% RSLogix 500 project LVD191219v4_Bot.RSS, saved by version 12.00.00.00 %
PROJECT "XLTCEBOT"    % processor: MicroLogix 1400 %

PROGRAM FILES
  LAD 2 "MAIN"  48 rungs  % Main Program Routine %
  LAD 4 "PACKAGER"  27 rungs  % normal %
  LAD 5 "NO PACKAGE"  7 rungs
  LAD 6 "TIMING"  11 rungs
  LAD 12 "ENABLES"  14 rungs
  LAD 14 "SPEED OUT"  14 rungs
  LAD 16 "TOTALCOUNT"  4 rungs
  LAD 18 "TESTTRIG1"  4 rungs
  LAD 20 "TESTTRIG2"  4 rungs
  LAD 24 "SKIPPED"  5 rungs
  LAD 70 "ALIGNFAILS"  4 rungs  % normal %
  LAD 80 "HSC BOT"  5 rungs
  LAD 100 "1 MS STI"  17 rungs  % high speed %
  LAD 102 "SPEED BOT"  8 rungs  % high speed %
  LAD 104 "P BOT"  7 rungs  % high speed %
  LAD 110 "SHIFT BOT"  7 rungs
  LAD 120 "OLDBOTOP"  7 rungs
  LAD 121 "OLDBOTOP"  8 rungs
  LAD 123 "BOTOPTIC"  2 rungs
  LAD 124 "BOTOPTIC"  4 rungs
  LAD 130 "INS1"  20 rungs
  LAD 131 "INS1RESULT"  7 rungs
  LAD 132 "INS1PASS"  5 rungs
  LAD 133 "INS1FAIL"  3 rungs
  LAD 134 "INS1ACQ"  8 rungs
  LAD 135 "Q1TIMETEST"  7 rungs
  LAD 136 "INS1TRIG"  6 rungs
  LAD 137 "FIFO1SET"  9 rungs
  LAD 138 "FIFO1GET"  8 rungs
  LAD 139 "INSDATA1"  3 rungs  % used for analysis %
  LAD 140 "TESTFAULT1"  9 rungs
  LAD 141 "INS1FIX1"  6 rungs
  LAD 142 "INS1FIX2"  3 rungs
  LAD 145 "INS2"  22 rungs
  LAD 146 "INS2RESULT"  7 rungs
  LAD 147 "INS2PASS"  5 rungs
  LAD 148 "INS2FAIL"  3 rungs
  LAD 149 "INS2ACQ"  8 rungs
  LAD 150 "Q2TIMETEST"  6 rungs
  LAD 151 "INS2TRIG"  5 rungs
  LAD 152 "FIFO2SET"  9 rungs
  LAD 153 "FIFO2GET"  8 rungs
  LAD 154 "INSDATA2"  3 rungs  % used for analysis %
  LAD 155 "TESTFAULT2"  9 rungs
  LAD 156 "INS2FIX1"  6 rungs
  LAD 157 "INS2FIX2"  3 rungs
  LAD 200 "XFEROUT"  9 rungs
  LAD 201 "XFER GOOD"  5 rungs
  LAD 202 "XFER NG"  5 rungs
  LAD 111, 122, 125, 144, 159: only END

DATA FILES
  O0 OUTPUT  11 elements
  I1 INPUT  11 elements
  S2 STATUS  66 elements
  B3 BINARY  64 elements
  T4 TIMER  40 elements
  C5 COUNTER  1 elements
  R6 CONTROL  20 elements
  N7 INTEGER  200 elements
  F8 FLOAT  100 elements
  B9 NU  256 elements
  B10 NU  1 elements
  B11 NU  256 elements
  B12 HMI_BINARY  22 elements  % general use with hmi to avoid additional reads %
  L13  COUNTS  256 elements
  F14 HMI_FLOATS  100 elements
  N15 HMI_INTS  100 elements
  L16 NU  100 elements
  B17 NU  128 elements
  B18 NU  128 elements
  L19 NU  10 elements
  L20 NU  10 elements
  L21 NU  10 elements
  L22 NU  10 elements
  L23 NU  100 elements
  L24 NU  100 elements
  L25 NU  10 elements
  L26 NU  10 elements
  L27 RATETIMES  50 elements  % Must have it's own file because it uses all 50 int %
  L28 INS1TIME  50 elements
  L29 INS1POS  50 elements
  L30 INS2TIME  50 elements
  L31 INS2POS  50 elements
  L42 COMS  52 elements
  RI43 RI1  11 elements
  MG44 MSG  11 elements
  B181 BLANK  256 elements  % used to wipe bs files %
  F182 TEST FLOAT  50 elements
  L183 TEST LONG  50 elements
  N184 TEST INTS  50 elements
  B185 TEST BITS  50 elements
  N186 HMI INTS  50 elements
  L187 HMI LONG  50 elements
  F188 HMI FLOAT  50 elements
  B189 HMI BITS  50 elements
  L190 COUNTS  50 elements
  B191 ERROR BITS  10 elements
  L192 SPD OFFSET  50 elements
  F193 SPD OFFSET  50 elements
  B194 BOT GOOD  128 elements
  B195 BOT NG  128 elements
  B196 CTRL BITS  50 elements
  N197 CTRL INTS  50 elements
  B198 TRK BITS  50 elements
  L199 TRK LONG  50 elements
  N200 TRK INTS  50 elements
  L201 INS LONG  50 elements
  B202 INS BITS  50 elements
  N203 INS INTS  50 elements
  L204 CTRL LONG  50 elements
  F205 CTRL FLTS  50 elements

LADDER 2 "MAIN"    % Main Program Routine %
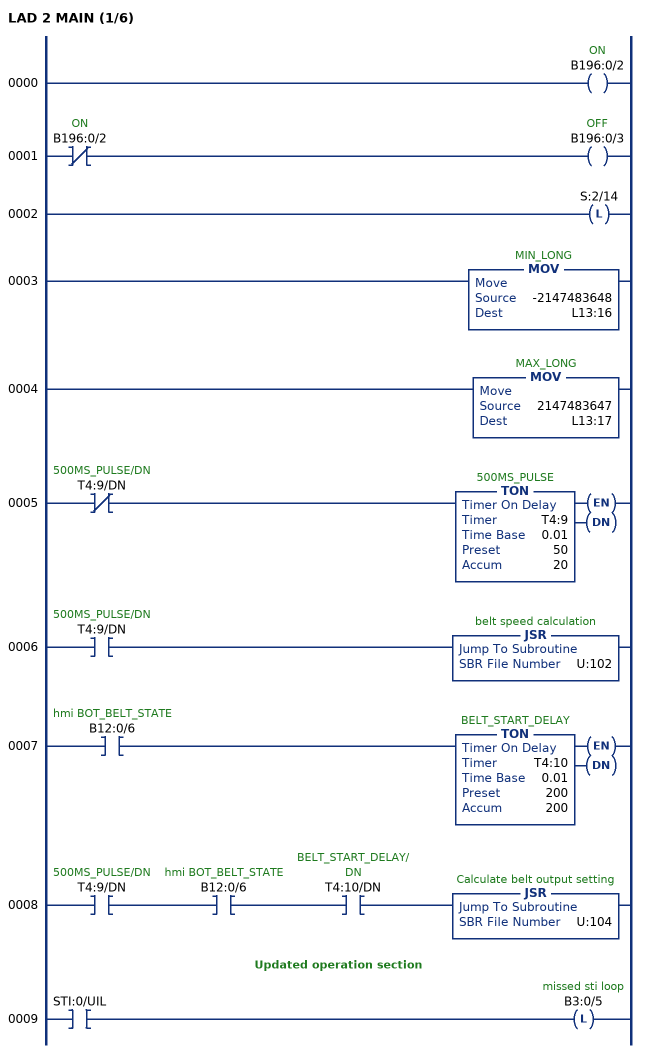
% Rung: 0 %
SOR OTE B196:0/2 EOR
%   B196:0/2  ON %
% Rung: 1 %
SOR XIO B196:0/2 OTE B196:0/3 EOR
%   B196:0/2  ON %
%   B196:0/3  OFF %
% Rung: 2 %
SOR OTL S:2/14 EOR
% Rung: 3 %
SOR MOV -2147483648 L13:16 EOR
%   L13:16  MIN_LONG %
% Rung: 4 %
SOR MOV 2147483647 L13:17 EOR
%   L13:17  MAX_LONG %
% Rung: 5 %
SOR XIO T4:9/DN TON T4:9 0.01 50 20 EOR
%   T4:9  500MS_PULSE %
% Rung: 6 %
SOR XIC T4:9/DN JSR U:102 EOR
%   T4:9  500MS_PULSE %
%   U:102  "belt speed calculation" %
% Rung: 7 %
SOR XIC B12:0/6 TON T4:10 0.01 200 200 EOR
%   B12:0/6  BOT_BELT_STATE  "hmi" %
%   T4:10  BELT_START_DELAY %
% Rung: 8 %
SOR XIC T4:9/DN XIC B12:0/6 XIC T4:10/DN JSR U:104 EOR
%   T4:9  500MS_PULSE %
%   B12:0/6  BOT_BELT_STATE  "hmi" %
%   T4:10  BELT_START_DELAY %
%   U:104  "Calculate belt output setting" %
% Rung: 9 %
% TITLE: Updated operation section %
SOR XIC STI:0/UIL OTL B3:0/5 EOR
%   B3:0/5  "missed sti loop" %

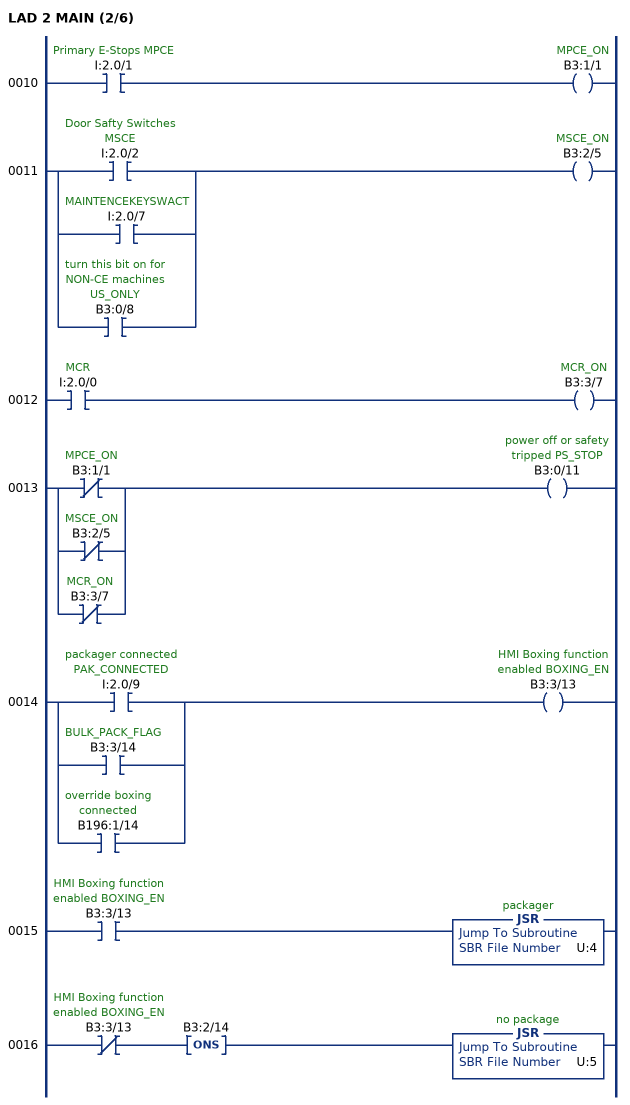
% Rung: 10 %
SOR XIC I:2.0/1 OTE B3:1/1 EOR
%   I:2.0/1  MPCE  "Primary E-Stops" %
%   B3:1/1  MPCE_ON %
% Rung: 11 %
SOR BST XIC I:2.0/2 NXB XIC I:2.0/7 NXB XIC B3:0/8 BND OTE B3:2/5 EOR
%   I:2.0/2  MSCE  "Door Safty Switches" %
%   I:2.0/7  MAINTENCEKEYSWACT %
%   B3:0/8  US_ONLY  "turn this bit on for NON-CE machines" %
%   B3:2/5  MSCE_ON %
% Rung: 12 %
SOR XIC I:2.0/0 OTE B3:3/7 EOR
%   I:2.0/0  MCR %
%   B3:3/7  MCR_ON %
% Rung: 13 %
SOR BST XIO B3:1/1 NXB XIO B3:2/5 NXB XIO B3:3/7 BND OTE B3:0/11 EOR
%   B3:1/1  MPCE_ON %
%   B3:2/5  MSCE_ON %
%   B3:3/7  MCR_ON %
%   B3:0/11  PS_STOP  "power off or safety tripped" %
% Rung: 14 %
SOR BST XIC I:2.0/9 NXB XIC B3:3/14 NXB XIC B196:1/14 BND OTE B3:3/13 EOR
%   I:2.0/9  PAK_CONNECTED  "packager connected" %
%   B3:3/14  BULK_PACK_FLAG %
%   B196:1/14  "override boxing connected" %
%   B3:3/13  BOXING_EN  "HMI Boxing function enabled" %
% Rung: 15 %
SOR XIC B3:3/13 JSR U:4 EOR
%   B3:3/13  BOXING_EN  "HMI Boxing function enabled" %
%   U:4  "packager" %
% Rung: 16 %
SOR XIO B3:3/13 ONS B3:2/14 JSR U:5 EOR
%   B3:3/13  BOXING_EN  "HMI Boxing function enabled" %
%   U:5  "no package" %

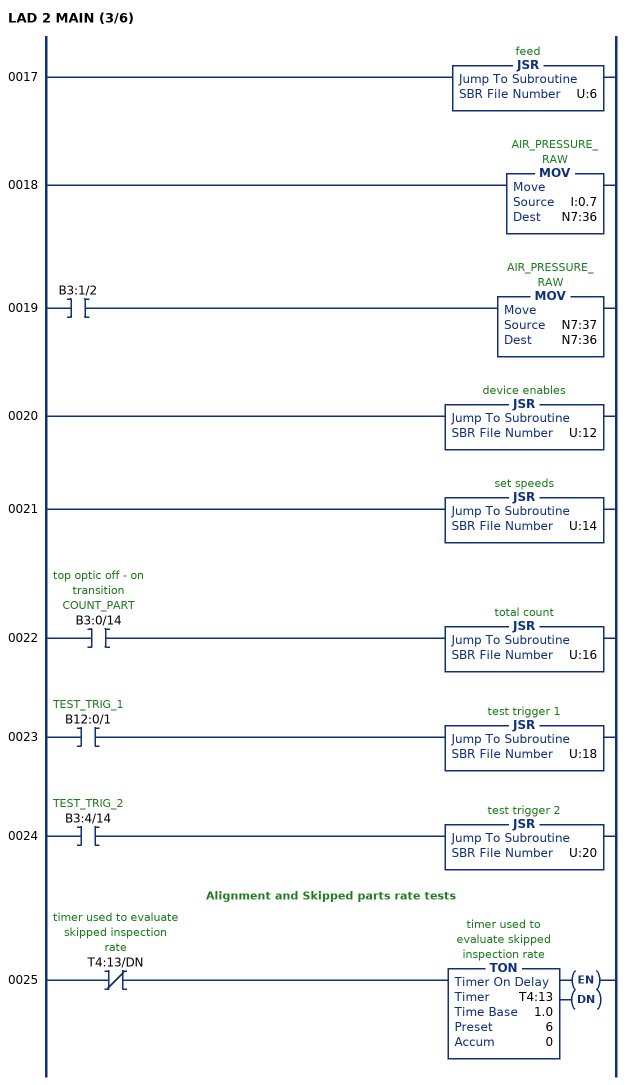
% Rung: 17 %
SOR JSR U:6 EOR
%   U:6  "feed" %
% Rung: 18 %
SOR MOV I:0.7 N7:36 EOR
%   I:0.7  AIR_PRESSURE  "Air Presure Sensor Input Signal" %
%   N7:36  AIR_PRESSURE_RAW %
% Rung: 19 %
SOR XIC B3:1/2 MOV N7:37 N7:36 EOR
%   N7:36  AIR_PRESSURE_RAW %
% Rung: 20 %
SOR JSR U:12 EOR
%   U:12  "device enables" %
% Rung: 21 %
SOR JSR U:14 EOR
%   U:14  "set speeds" %
% Rung: 22 %
SOR XIC B3:0/14 JSR U:16 EOR
%   B3:0/14  COUNT_PART  "top optic off - on transition" %
%   U:16  "total count" %
% Rung: 23 %
SOR XIC B12:0/1 JSR U:18 EOR
%   B12:0/1  TEST_TRIG_1 %
%   U:18  "test trigger 1" %
% Rung: 24 %
SOR XIC B3:4/14 JSR U:20 EOR
%   B3:4/14  TEST_TRIG_2 %
%   U:20  "test trigger 2" %
% Rung: 25 %
% TITLE: Alignment and Skipped parts rate tests %
SOR XIO T4:13/DN TON T4:13 1.0 6 0 EOR
%   T4:13  "timer used to evaluate skipped inspection rate" %

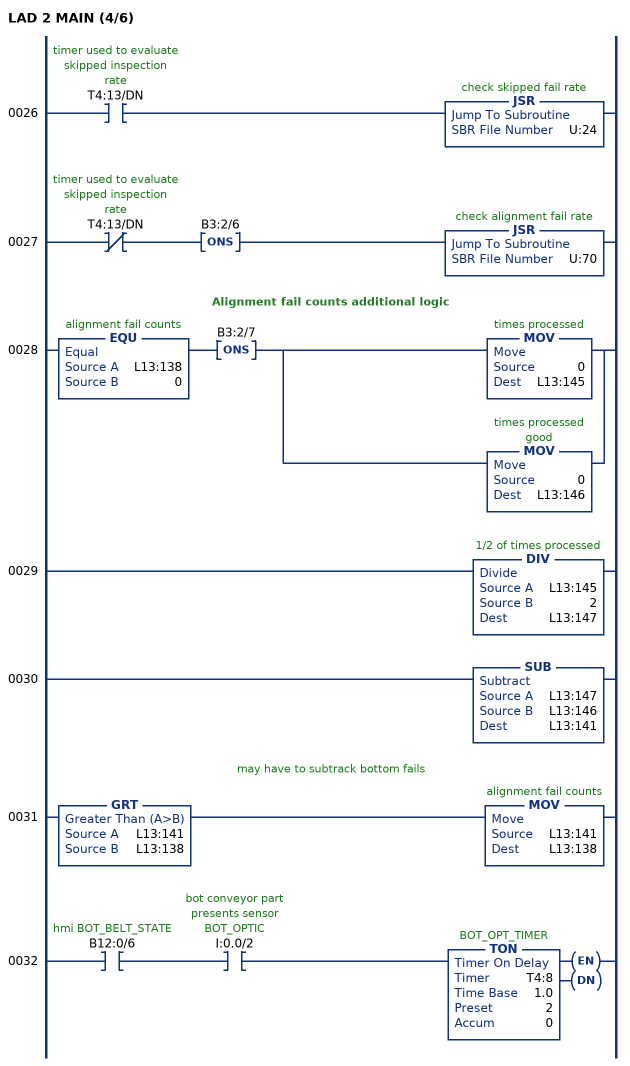
% Rung: 26 %
SOR XIC T4:13/DN JSR U:24 EOR
%   T4:13  "timer used to evaluate skipped inspection rate" %
%   U:24  "check skipped fail rate" %
% Rung: 27 %
SOR XIO T4:13/DN ONS B3:2/6 JSR U:70 EOR
%   T4:13  "timer used to evaluate skipped inspection rate" %
%   U:70  "check alignment fail rate" %
% Rung: 28 %
% TITLE: Alignment fail counts additional logic %
SOR EQU L13:138 0 ONS B3:2/7 BST MOV 0 L13:145 NXB MOV 0 L13:146 BND EOR
%   L13:138  "alignment fail counts" %
%   L13:145  "times processed" %
%   L13:146  "times processed good" %
% Rung: 29 %
SOR DIV L13:145 2 L13:147 EOR
%   L13:145  "times processed" %
%   L13:147  "1/2 of times processed" %
% Rung: 30 %
SOR SUB L13:147 L13:146 L13:141 EOR
%   L13:147  "1/2 of times processed" %
%   L13:146  "times processed good" %
% Rung: 31 %
% may have to subtrack bottom fails %
SOR GRT L13:141 L13:138 MOV L13:141 L13:138 EOR
%   L13:138  "alignment fail counts" %
% Rung: 32 %
SOR XIC B12:0/6 XIC I:0.0/2 TON T4:8 1.0 2 0 EOR
%   B12:0/6  BOT_BELT_STATE  "hmi" %
%   I:0.0/2  BOT_OPTIC  "bot conveyor part presents sensor" %
%   T4:8  BOT_OPT_TIMER %

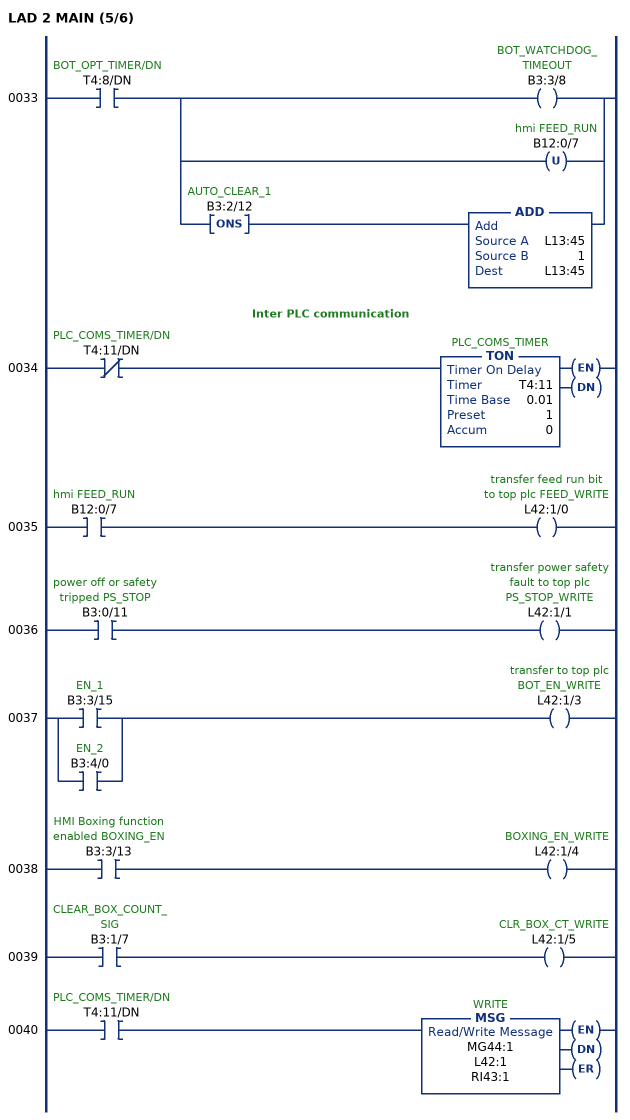
% Rung: 33 %
SOR XIC T4:8/DN BST OTE B3:3/8 NXB OTU B12:0/7 NXB ONS B3:2/12 ADD L13:45 1 L13:45 BND EOR
%   T4:8  BOT_OPT_TIMER %
%   B3:3/8  BOT_WATCHDOG_TIMEOUT %
%   B12:0/7  FEED_RUN  "hmi" %
%   B3:2/12  AUTO_CLEAR_1 %
% Rung: 34 %
% TITLE: Inter PLC communication %
SOR XIO T4:11/DN TON T4:11 0.01 1 0 EOR
%   T4:11  PLC_COMS_TIMER %
% Rung: 35 %
SOR XIC B12:0/7 OTE L42:1/0 EOR
%   B12:0/7  FEED_RUN  "hmi" %
%   L42:1/0  FEED_WRITE  "transfer feed run bit to top plc" %
% Rung: 36 %
SOR XIC B3:0/11 OTE L42:1/1 EOR
%   B3:0/11  PS_STOP  "power off or safety tripped" %
%   L42:1/1  PS_STOP_WRITE  "transfer power safety fault to top plc" %
% Rung: 37 %
SOR BST XIC B3:3/15 NXB XIC B3:4/0 BND OTE L42:1/3 EOR
%   B3:3/15  EN_1 %
%   B3:4/0  EN_2 %
%   L42:1/3  BOT_EN_WRITE  "transfer to top plc" %
% Rung: 38 %
SOR XIC B3:3/13 OTE L42:1/4 EOR
%   B3:3/13  BOXING_EN  "HMI Boxing function enabled" %
%   L42:1/4  BOXING_EN_WRITE %
% Rung: 39 %
SOR XIC B3:1/7 OTE L42:1/5 EOR
%   B3:1/7  CLEAR_BOX_COUNT_SIG %
%   L42:1/5  CLR_BOX_CT_WRITE %
% Rung: 40 %
SOR XIC T4:11/DN MSG MG44:1 L42:1 RI43:1 EOR
%   T4:11  PLC_COMS_TIMER %
%   MSG set-up: 500CPU Write | 33 | 1 | L42:0 | L42:1 | 0 | 0 | 0 | 192.168.222.101:0 | 0 | 0 | 192.168.222.101 | RI43:1 %
%   MG44:1  WRITE %
%   L42:1  WRITE_BITS %

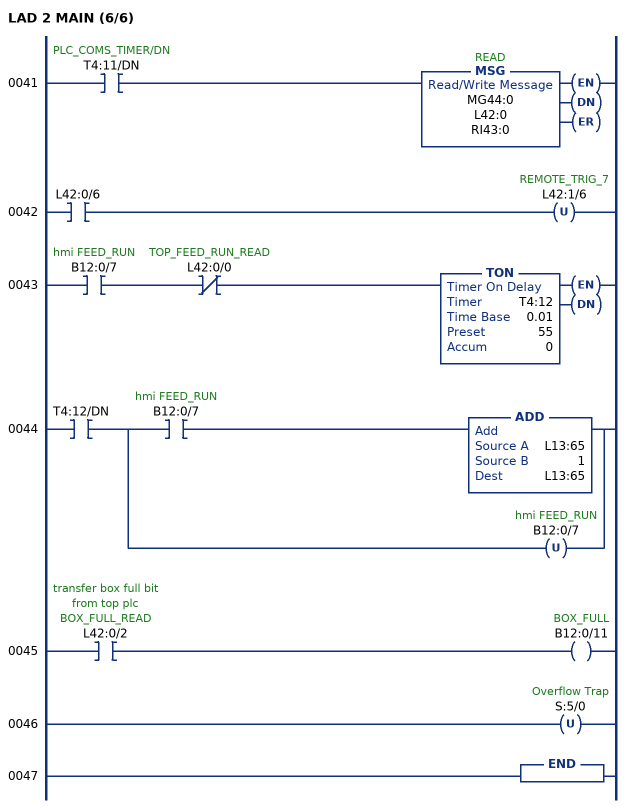
% Rung: 41 %
SOR XIC T4:11/DN MSG MG44:0 L42:0 RI43:0 EOR
%   T4:11  PLC_COMS_TIMER %
%   MSG set-up: 500CPU Read | 33 | 1 | L42:1 | L42:0 | 0 | 0 | 0 | 192.168.222.101:0 | 0 | 0 | 192.168.222.101 | RI43:0 %
%   MG44:0  READ %
%   L42:0  READ_BITS %
% Rung: 42 %
SOR XIC L42:0/6 OTU L42:1/6 EOR
%   L42:1/6  REMOTE_TRIG_7 %
% Rung: 43 %
SOR XIC B12:0/7 XIO L42:0/0 TON T4:12 0.01 55 0 EOR
%   B12:0/7  FEED_RUN  "hmi" %
%   L42:0/0  TOP_FEED_RUN_READ %
% Rung: 44 %
SOR XIC T4:12/DN BST XIC B12:0/7 ADD L13:65 1 L13:65 NXB OTU B12:0/7 BND EOR
%   B12:0/7  FEED_RUN  "hmi" %
% Rung: 45 %
SOR XIC L42:0/2 OTE B12:0/11 EOR
%   L42:0/2  BOX_FULL_READ  "transfer box full bit from top plc" %
%   B12:0/11  BOX_FULL %
% Rung: 46 %
SOR OTU S:5/0 EOR
%   S:5/0  "Overflow Trap" %
% Rung: 47 %
SOR END EOR

LADDER 4 "PACKAGER"    % normal %
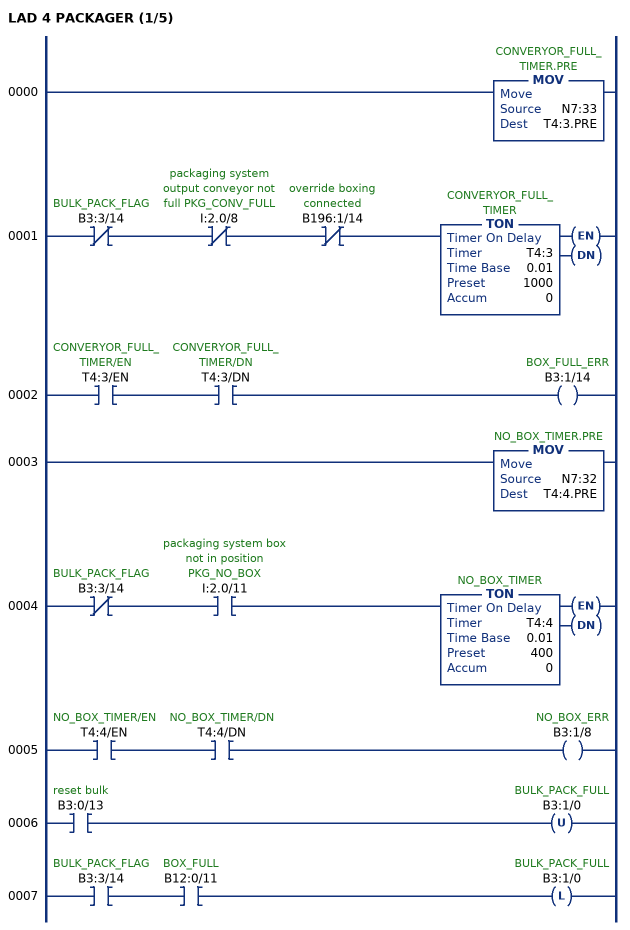
% Rung: 0 %
SOR MOV N7:33 T4:3.PRE EOR
%   T4:3  CONVERYOR_FULL_TIMER %
% Rung: 1 %
SOR XIO B3:3/14 XIO I:2.0/8 XIO B196:1/14 TON T4:3 0.01 1000 0 EOR
%   B3:3/14  BULK_PACK_FLAG %
%   I:2.0/8  PKG_CONV_FULL  "packaging system output conveyor not full" %
%   B196:1/14  "override boxing connected" %
%   T4:3  CONVERYOR_FULL_TIMER %
% Rung: 2 %
SOR XIC T4:3/EN XIC T4:3/DN OTE B3:1/14 EOR
%   T4:3  CONVERYOR_FULL_TIMER %
%   B3:1/14  BOX_FULL_ERR %
% Rung: 3 %
SOR MOV N7:32 T4:4.PRE EOR
%   T4:4  NO_BOX_TIMER %
% Rung: 4 %
SOR XIO B3:3/14 XIC I:2.0/11 TON T4:4 0.01 400 0 EOR
%   B3:3/14  BULK_PACK_FLAG %
%   I:2.0/11  PKG_NO_BOX  "packaging system box not in position" %
%   T4:4  NO_BOX_TIMER %
% Rung: 5 %
SOR XIC T4:4/EN XIC T4:4/DN OTE B3:1/8 EOR
%   T4:4  NO_BOX_TIMER %
%   B3:1/8  NO_BOX_ERR %
% Rung: 6 %
SOR XIC B3:0/13 OTU B3:1/0 EOR
%   B3:0/13  "reset bulk" %
%   B3:1/0  BULK_PACK_FULL %
% Rung: 7 %
SOR XIC B3:3/14 XIC B12:0/11 OTL B3:1/0 EOR
%   B3:3/14  BULK_PACK_FLAG %
%   B12:0/11  BOX_FULL %
%   B3:1/0  BULK_PACK_FULL %

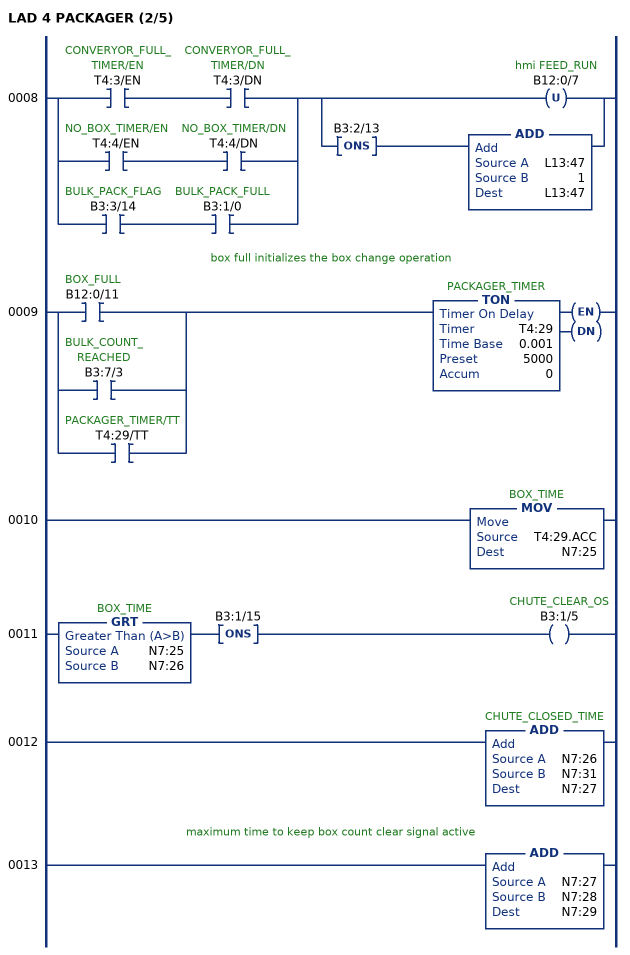
% Rung: 8 %
SOR BST XIC T4:3/EN XIC T4:3/DN NXB XIC T4:4/EN XIC T4:4/DN NXB XIC B3:3/14 XIC B3:1/0 BND BST OTU B12:0/7 NXB ONS B3:2/13 ADD L13:47 1 L13:47 BND EOR
%   T4:3  CONVERYOR_FULL_TIMER %
%   T4:4  NO_BOX_TIMER %
%   B3:3/14  BULK_PACK_FLAG %
%   B3:1/0  BULK_PACK_FULL %
%   B12:0/7  FEED_RUN  "hmi" %
% Rung: 9 %
% box full initializes the box change operation %
SOR BST XIC B12:0/11 NXB XIC B3:7/3 NXB XIC T4:29/TT BND TON T4:29 0.001 5000 0 EOR
%   B12:0/11  BOX_FULL %
%   B3:7/3  BULK_COUNT_REACHED %
%   T4:29  PACKAGER_TIMER %
% Rung: 10 %
SOR MOV T4:29.ACC N7:25 EOR
%   T4:29  PACKAGER_TIMER %
%   N7:25  BOX_TIME %
% Rung: 11 %
SOR GRT N7:25 N7:26 ONS B3:1/15 OTE B3:1/5 EOR
%   N7:25  BOX_TIME %
%   N7:26  CHUTE_CLEAR_TIME %
%   B3:1/5  CHUTE_CLEAR_OS %
% Rung: 12 %
SOR ADD N7:26 N7:31 N7:27 EOR
%   N7:26  CHUTE_CLEAR_TIME %
%   N7:27  CHUTE_CLOSED_TIME %
% Rung: 13 %
% maximum time to keep box count clear signal active %
SOR ADD N7:27 N7:28 N7:29 EOR
%   N7:27  CHUTE_CLOSED_TIME %

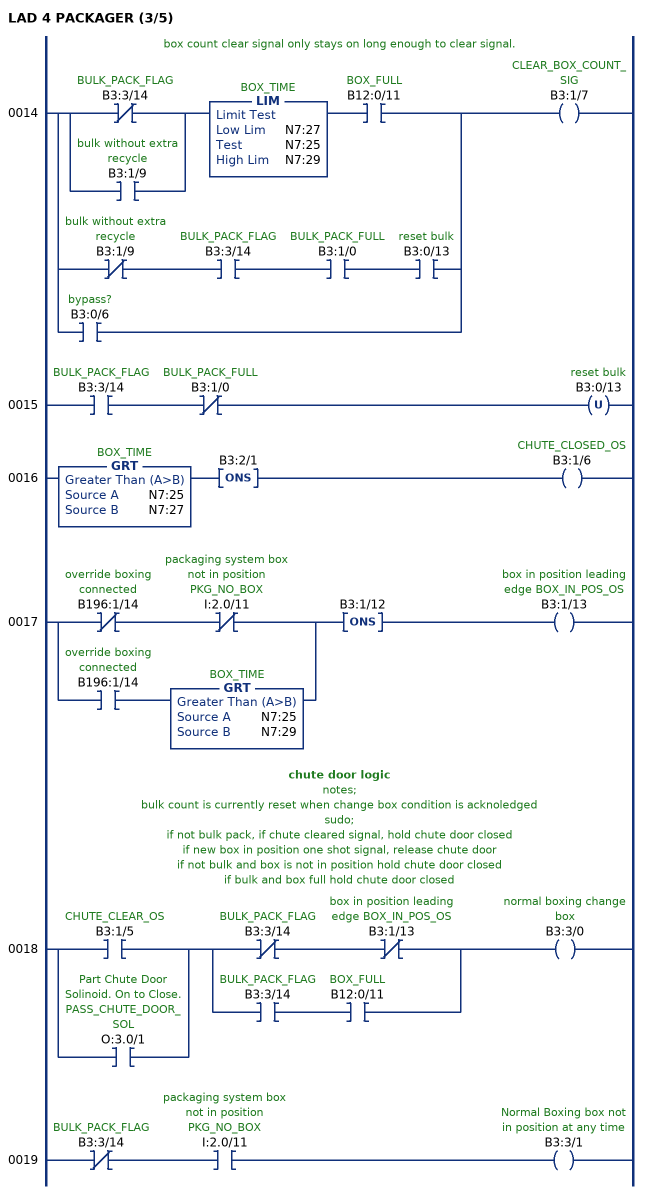
% Rung: 14 %
% box count clear signal only stays on long enough to clear signal. %
SOR BST BST XIO B3:3/14 NXB XIC B3:1/9 BND LIM N7:27 N7:25 N7:29 XIC B12:0/11 NXB XIO B3:1/9 XIC B3:3/14 XIC B3:1/0 XIC B3:0/13 NXB XIC B3:0/6 BND OTE B3:1/7 EOR
%   B3:3/14  BULK_PACK_FLAG %
%   B3:1/9  "bulk without extra recycle" %
%   N7:27  CHUTE_CLOSED_TIME %
%   N7:25  BOX_TIME %
%   B12:0/11  BOX_FULL %
%   B3:1/0  BULK_PACK_FULL %
%   B3:0/13  "reset bulk" %
%   B3:0/6  "bypass?" %
%   B3:1/7  CLEAR_BOX_COUNT_SIG %
% Rung: 15 %
SOR XIC B3:3/14 XIO B3:1/0 OTU B3:0/13 EOR
%   B3:3/14  BULK_PACK_FLAG %
%   B3:1/0  BULK_PACK_FULL %
%   B3:0/13  "reset bulk" %
% Rung: 16 %
SOR GRT N7:25 N7:27 ONS B3:2/1 OTE B3:1/6 EOR
%   N7:25  BOX_TIME %
%   N7:27  CHUTE_CLOSED_TIME %
%   B3:1/6  CHUTE_CLOSED_OS %
% Rung: 17 %
SOR BST XIO B196:1/14 XIO I:2.0/11 NXB XIC B196:1/14 GRT N7:25 N7:29 BND ONS B3:1/12 OTE B3:1/13 EOR
%   B196:1/14  "override boxing connected" %
%   I:2.0/11  PKG_NO_BOX  "packaging system box not in position" %
%   N7:25  BOX_TIME %
%   B3:1/13  BOX_IN_POS_OS  "box in position leading edge" %
% Rung: 18 %
% TITLE: chute door logic %
% notes;
% bulk count is currently reset when change box condition is acknoledged
% 
% sudo;
% if not bulk pack, if chute cleared signal, hold chute door closed
%           if new box in position one shot signal, release chute door
% if not bulk and box is not in position hold chute door closed
% if bulk and box full hold chute door closed %
SOR BST XIC B3:1/5 NXB XIC O:3.0/1 BND BST XIO B3:3/14 XIO B3:1/13 NXB XIC B3:3/14 XIC B12:0/11 BND OTE B3:3/0 EOR
%   B3:1/5  CHUTE_CLEAR_OS %
%   O:3.0/1  PASS_CHUTE_DOOR_SOL  "Part Chute Door Solinoid. On to Close." %
%   B3:3/14  BULK_PACK_FLAG %
%   B3:1/13  BOX_IN_POS_OS  "box in position leading edge" %
%   B12:0/11  BOX_FULL %
%   B3:3/0  "normal boxing change box" %
% Rung: 19 %
SOR XIO B3:3/14 XIC I:2.0/11 OTE B3:3/1 EOR
%   B3:3/14  BULK_PACK_FLAG %
%   I:2.0/11  PKG_NO_BOX  "packaging system box not in position" %
%   B3:3/1  "Normal Boxing box not in position at any time" %

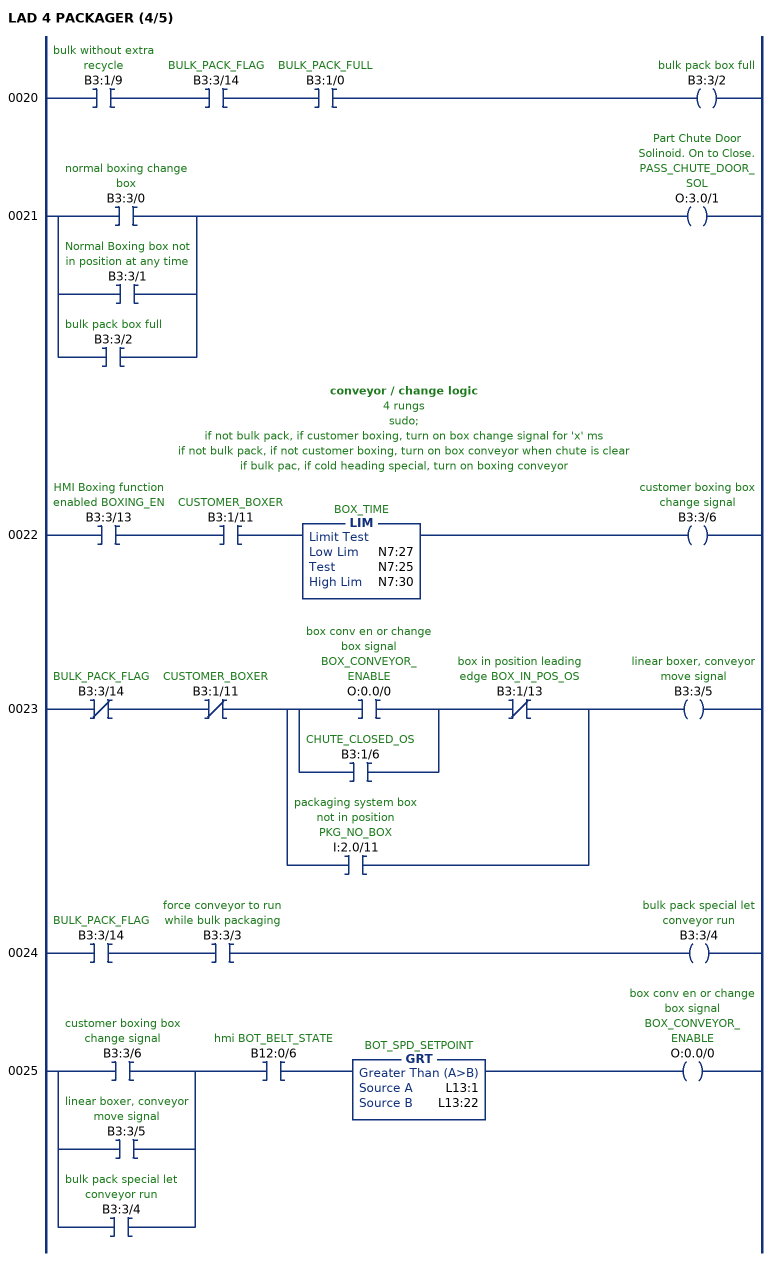
% Rung: 20 %
SOR XIC B3:1/9 XIC B3:3/14 XIC B3:1/0 OTE B3:3/2 EOR
%   B3:1/9  "bulk without extra recycle" %
%   B3:3/14  BULK_PACK_FLAG %
%   B3:1/0  BULK_PACK_FULL %
%   B3:3/2  "bulk pack box full" %
% Rung: 21 %
SOR BST XIC B3:3/0 NXB XIC B3:3/1 NXB XIC B3:3/2 BND OTE O:3.0/1 EOR
%   B3:3/0  "normal boxing change box" %
%   B3:3/1  "Normal Boxing box not in position at any time" %
%   B3:3/2  "bulk pack box full" %
%   O:3.0/1  PASS_CHUTE_DOOR_SOL  "Part Chute Door Solinoid. On to Close." %
% Rung: 22 %
% TITLE: conveyor / change logic %
% 4 rungs
% sudo;
% if not bulk pack, if customer boxing, turn on box change signal for 'x' ms
% if not bulk pack, if not customer boxing, turn on box conveyor when chute is clear
% if bulk pac, if cold heading special, turn on boxing conveyor %
SOR XIC B3:3/13 XIC B3:1/11 LIM N7:27 N7:25 N7:30 OTE B3:3/6 EOR
%   B3:3/13  BOXING_EN  "HMI Boxing function enabled" %
%   B3:1/11  CUSTOMER_BOXER %
%   N7:27  CHUTE_CLOSED_TIME %
%   N7:25  BOX_TIME %
%   N7:30  END_OF_CHANGE_SIG %
%   B3:3/6  "customer boxing box change signal" %
% Rung: 23 %
SOR XIO B3:3/14 XIO B3:1/11 BST BST XIC O:0.0/0 NXB XIC B3:1/6 BND XIO B3:1/13 NXB XIC I:2.0/11 BND OTE B3:3/5 EOR
%   B3:3/14  BULK_PACK_FLAG %
%   B3:1/11  CUSTOMER_BOXER %
%   O:0.0/0  BOX_CONVEYOR_ENABLE  "box conv en or change box signal" %
%   B3:1/6  CHUTE_CLOSED_OS %
%   B3:1/13  BOX_IN_POS_OS  "box in position leading edge" %
%   I:2.0/11  PKG_NO_BOX  "packaging system box not in position" %
%   B3:3/5  "linear boxer, conveyor move signal" %
% Rung: 24 %
SOR XIC B3:3/14 XIC B3:3/3 OTE B3:3/4 EOR
%   B3:3/14  BULK_PACK_FLAG %
%   B3:3/3  "force conveyor to run while bulk packaging" %
%   B3:3/4  "bulk pack special let conveyor run" %
% Rung: 25 %
SOR BST XIC B3:3/6 NXB XIC B3:3/5 NXB XIC B3:3/4 BND XIC B12:0/6 GRT L13:1 L13:22 OTE O:0.0/0 EOR
%   B3:3/6  "customer boxing box change signal" %
%   B3:3/5  "linear boxer, conveyor move signal" %
%   B3:3/4  "bulk pack special let conveyor run" %
%   B12:0/6  BOT_BELT_STATE  "hmi" %
%   L13:1  BOT_SPD_SETPOINT %
%   O:0.0/0  BOX_CONVEYOR_ENABLE  "box conv en or change box signal" %

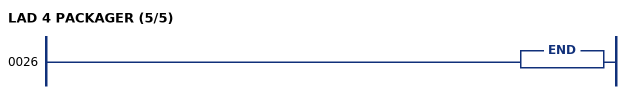
% Rung: 26 %
SOR END EOR

LADDER 5 "NO PACKAGE"
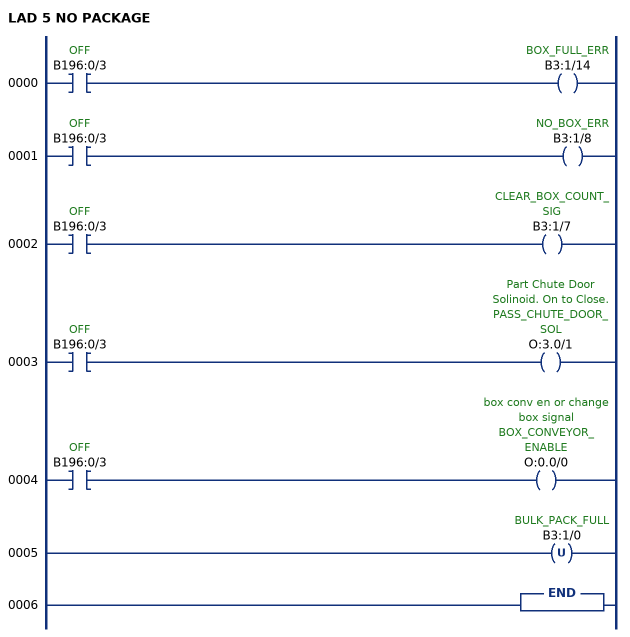
% Rung: 0 %
SOR XIC B196:0/3 OTE B3:1/14 EOR
%   B196:0/3  OFF %
%   B3:1/14  BOX_FULL_ERR %
% Rung: 1 %
SOR XIC B196:0/3 OTE B3:1/8 EOR
%   B196:0/3  OFF %
%   B3:1/8  NO_BOX_ERR %
% Rung: 2 %
SOR XIC B196:0/3 OTE B3:1/7 EOR
%   B196:0/3  OFF %
%   B3:1/7  CLEAR_BOX_COUNT_SIG %
% Rung: 3 %
SOR XIC B196:0/3 OTE O:3.0/1 EOR
%   B196:0/3  OFF %
%   O:3.0/1  PASS_CHUTE_DOOR_SOL  "Part Chute Door Solinoid. On to Close." %
% Rung: 4 %
SOR XIC B196:0/3 OTE O:0.0/0 EOR
%   B196:0/3  OFF %
%   O:0.0/0  BOX_CONVEYOR_ENABLE  "box conv en or change box signal" %
% Rung: 5 %
SOR OTU B3:1/0 EOR
%   B3:1/0  BULK_PACK_FULL %
% Rung: 6 %
SOR END EOR

LADDER 6 "TIMING"
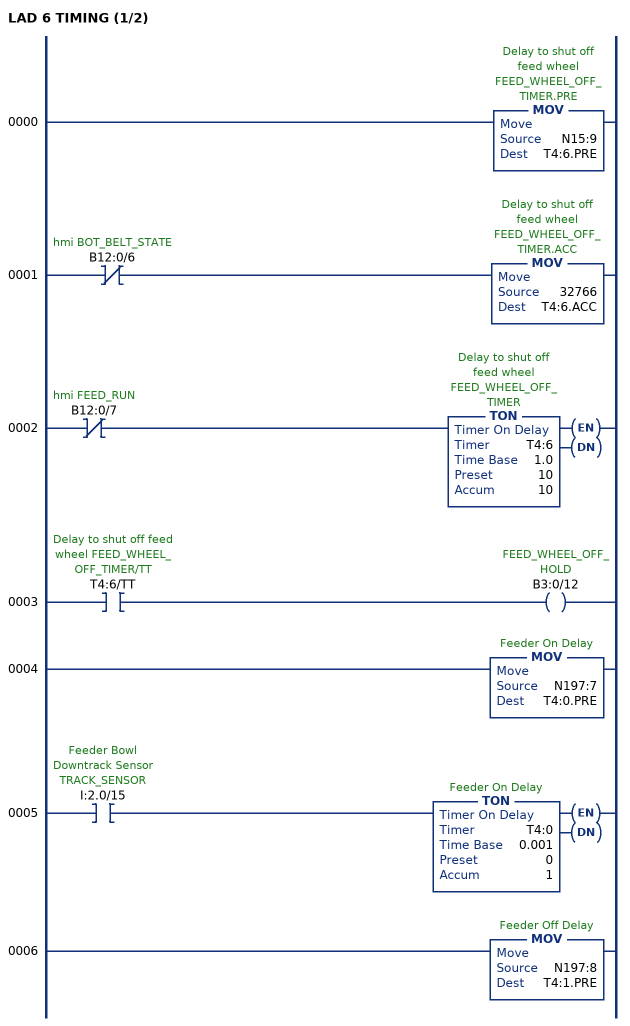
% Rung: 0 %
SOR MOV N15:9 T4:6.PRE EOR
%   N15:9  FEED_WHEEL_STOP_TIME %
%   T4:6  FEED_WHEEL_OFF_TIMER  "Delay to shut off feed wheel" %
% Rung: 1 %
SOR XIO B12:0/6 MOV 32766 T4:6.ACC EOR
%   B12:0/6  BOT_BELT_STATE  "hmi" %
%   T4:6  FEED_WHEEL_OFF_TIMER  "Delay to shut off feed wheel" %
% Rung: 2 %
SOR XIO B12:0/7 TON T4:6 1.0 10 10 EOR
%   B12:0/7  FEED_RUN  "hmi" %
%   T4:6  FEED_WHEEL_OFF_TIMER  "Delay to shut off feed wheel" %
% Rung: 3 %
SOR XIC T4:6/TT OTE B3:0/12 EOR
%   T4:6  FEED_WHEEL_OFF_TIMER  "Delay to shut off feed wheel" %
%   B3:0/12  FEED_WHEEL_OFF_HOLD %
% Rung: 4 %
SOR MOV N197:7 T4:0.PRE EOR
%   N197:7  "down track on delay" %
%   T4:0  "Feeder On Delay" %
% Rung: 5 %
SOR XIC I:2.0/15 TON T4:0 0.001 0 1 EOR
%   I:2.0/15  TRACK_SENSOR  "Feeder Bowl Downtrack Sensor" %
%   T4:0  "Feeder On Delay" %
% Rung: 6 %
SOR MOV N197:8 T4:1.PRE EOR
%   N197:8  "down track off delay" %
%   T4:1  "Feeder Off Delay" %

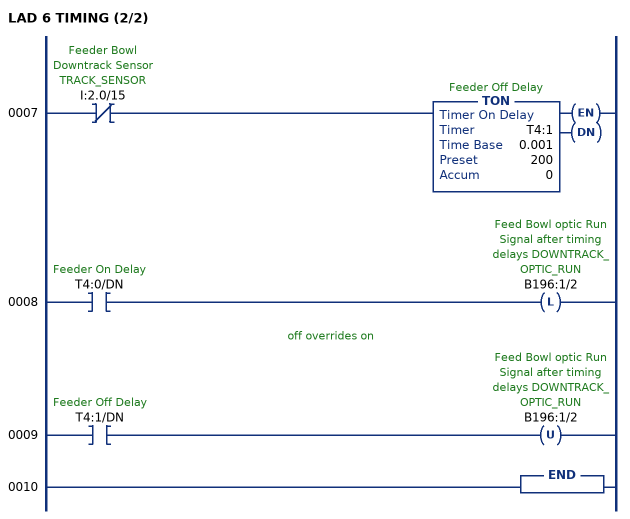
% Rung: 7 %
SOR XIO I:2.0/15 TON T4:1 0.001 200 0 EOR
%   I:2.0/15  TRACK_SENSOR  "Feeder Bowl Downtrack Sensor" %
%   T4:1  "Feeder Off Delay" %
% Rung: 8 %
SOR XIC T4:0/DN OTL B196:1/2 EOR
%   T4:0  "Feeder On Delay" %
%   B196:1/2  DOWNTRACK_OPTIC_RUN  "Feed Bowl optic Run Signal after timing delays" %
% Rung: 9 %
% off overrides on %
SOR XIC T4:1/DN OTU B196:1/2 EOR
%   T4:1  "Feeder Off Delay" %
%   B196:1/2  DOWNTRACK_OPTIC_RUN  "Feed Bowl optic Run Signal after timing delays" %
% Rung: 10 %
SOR END EOR

LADDER 12 "ENABLES"
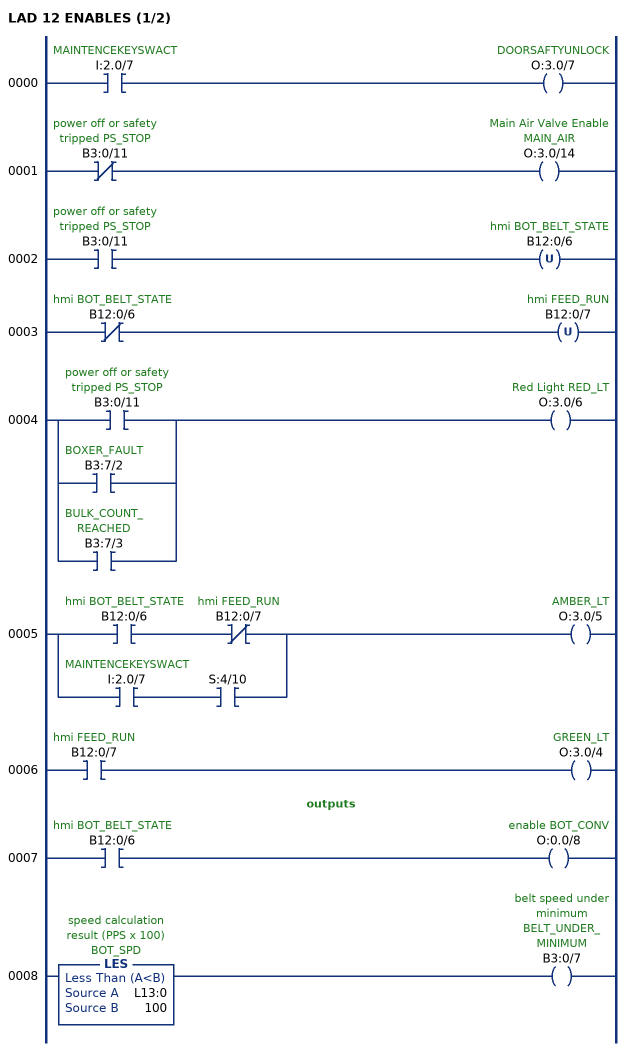
% Rung: 0 %
SOR XIC I:2.0/7 OTE O:3.0/7 EOR
%   I:2.0/7  MAINTENCEKEYSWACT %
%   O:3.0/7  DOORSAFTYUNLOCK %
% Rung: 1 %
SOR XIO B3:0/11 OTE O:3.0/14 EOR
%   B3:0/11  PS_STOP  "power off or safety tripped" %
%   O:3.0/14  MAIN_AIR  "Main Air Valve Enable" %
% Rung: 2 %
SOR XIC B3:0/11 OTU B12:0/6 EOR
%   B3:0/11  PS_STOP  "power off or safety tripped" %
%   B12:0/6  BOT_BELT_STATE  "hmi" %
% Rung: 3 %
SOR XIO B12:0/6 OTU B12:0/7 EOR
%   B12:0/6  BOT_BELT_STATE  "hmi" %
%   B12:0/7  FEED_RUN  "hmi" %
% Rung: 4 %
SOR BST XIC B3:0/11 NXB XIC B3:7/2 NXB XIC B3:7/3 BND OTE O:3.0/6 EOR
%   B3:0/11  PS_STOP  "power off or safety tripped" %
%   B3:7/2  BOXER_FAULT %
%   B3:7/3  BULK_COUNT_REACHED %
%   O:3.0/6  RED_LT  "Red Light" %
% Rung: 5 %
SOR BST XIC B12:0/6 XIO B12:0/7 NXB XIC I:2.0/7 XIC S:4/10 BND OTE O:3.0/5 EOR
%   B12:0/6  BOT_BELT_STATE  "hmi" %
%   B12:0/7  FEED_RUN  "hmi" %
%   I:2.0/7  MAINTENCEKEYSWACT %
%   O:3.0/5  AMBER_LT %
% Rung: 6 %
SOR XIC B12:0/7 OTE O:3.0/4 EOR
%   B12:0/7  FEED_RUN  "hmi" %
%   O:3.0/4  GREEN_LT %
% Rung: 7 %
% TITLE: outputs %
SOR XIC B12:0/6 OTE O:0.0/8 EOR
%   B12:0/6  BOT_BELT_STATE  "hmi" %
%   O:0.0/8  BOT_CONV  "enable" %
% Rung: 8 %
SOR LES L13:0 100 OTE B3:0/7 EOR
%   L13:0  BOT_SPD  "speed calculation result (PPS x 100)" %
%   B3:0/7  BELT_UNDER_MINIMUM  "belt speed under minimum" %

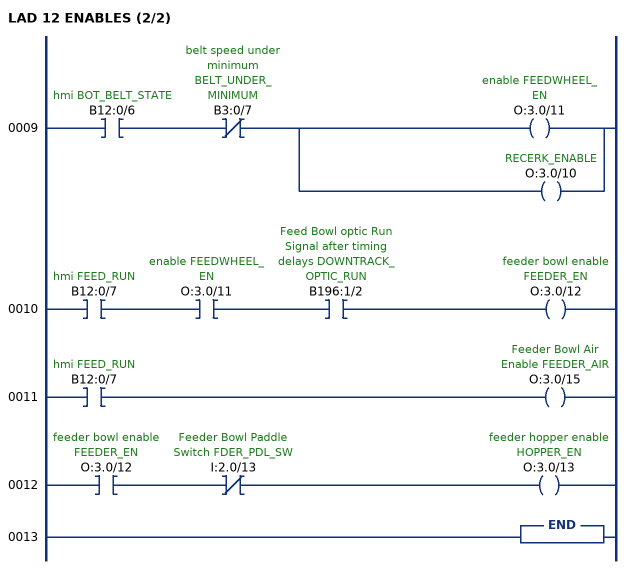
% Rung: 9 %
SOR XIC B12:0/6 XIO B3:0/7 BST OTE O:3.0/11 NXB OTE O:3.0/10 BND EOR
%   B12:0/6  BOT_BELT_STATE  "hmi" %
%   B3:0/7  BELT_UNDER_MINIMUM  "belt speed under minimum" %
%   O:3.0/11  FEEDWHEEL_EN  "enable" %
%   O:3.0/10  RECERK_ENABLE %
% Rung: 10 %
SOR XIC B12:0/7 XIC O:3.0/11 XIC B196:1/2 OTE O:3.0/12 EOR
%   B12:0/7  FEED_RUN  "hmi" %
%   O:3.0/11  FEEDWHEEL_EN  "enable" %
%   B196:1/2  DOWNTRACK_OPTIC_RUN  "Feed Bowl optic Run Signal after timing delays" %
%   O:3.0/12  FEEDER_EN  "feeder bowl enable" %
% Rung: 11 %
SOR XIC B12:0/7 OTE O:3.0/15 EOR
%   B12:0/7  FEED_RUN  "hmi" %
%   O:3.0/15  FEEDER_AIR  "Feeder Bowl Air Enable" %
% Rung: 12 %
SOR XIC O:3.0/12 XIO I:2.0/13 OTE O:3.0/13 EOR
%   O:3.0/12  FEEDER_EN  "feeder bowl enable" %
%   I:2.0/13  FDER_PDL_SW  "Feeder Bowl Paddle Switch" %
%   O:3.0/13  HOPPER_EN  "feeder hopper enable" %
% Rung: 13 %
SOR END EOR

LADDER 14 "SPEED OUT"
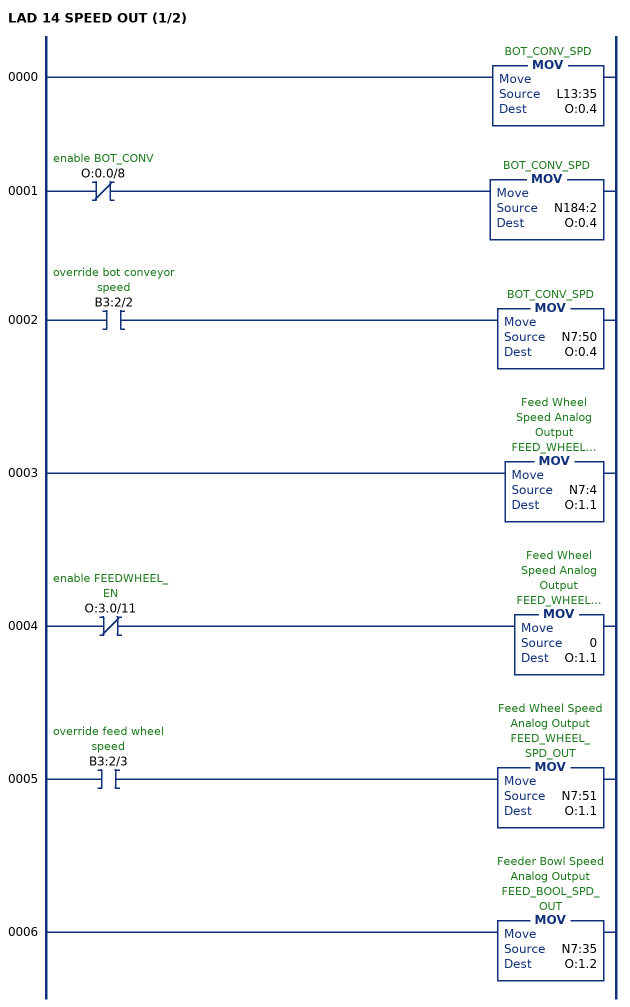
% Rung: 0 %
SOR MOV L13:35 O:0.4 EOR
%   L13:35  SCALED_BOT_VALUE %
%   O:0.4  BOT_CONV_SPD %
% Rung: 1 %
SOR XIO O:0.0/8 MOV N184:2 O:0.4 EOR
%   O:0.0/8  BOT_CONV  "enable" %
%   O:0.4  BOT_CONV_SPD %
% Rung: 2 %
SOR XIC B3:2/2 MOV N7:50 O:0.4 EOR
%   B3:2/2  "override bot conveyor speed" %
%   O:0.4  BOT_CONV_SPD %
% Rung: 3 %
SOR MOV N7:4 O:1.1 EOR
%   N7:4  FEED_WHEEL_SPD  "Feed Wheel Speed" %
%   O:1.1  FEED_WHEEL_SPD_OUT  "Feed Wheel Speed Analog Output" %
% Rung: 4 %
SOR XIO O:3.0/11 MOV 0 O:1.1 EOR
%   O:3.0/11  FEEDWHEEL_EN  "enable" %
%   O:1.1  FEED_WHEEL_SPD_OUT  "Feed Wheel Speed Analog Output" %
% Rung: 5 %
SOR XIC B3:2/3 MOV N7:51 O:1.1 EOR
%   B3:2/3  "override feed wheel speed" %
%   O:1.1  FEED_WHEEL_SPD_OUT  "Feed Wheel Speed Analog Output" %
% Rung: 6 %
SOR MOV N7:35 O:1.2 EOR
%   N7:35  FEEDER_SPD %
%   O:1.2  FEED_BOOL_SPD_OUT  "Feeder Bowl Speed Analog Output" %

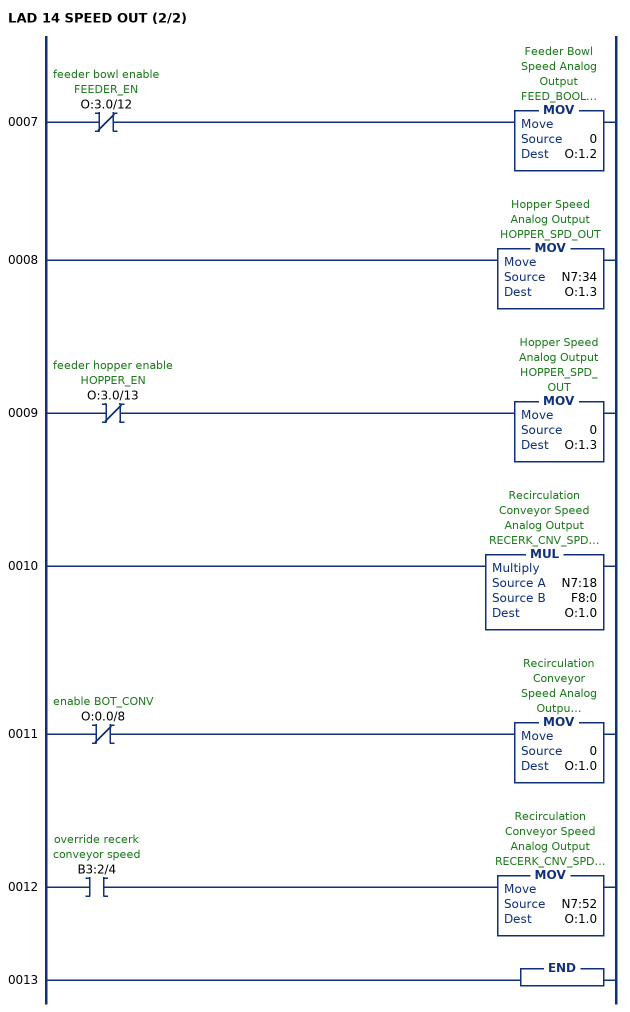
% Rung: 7 %
SOR XIO O:3.0/12 MOV 0 O:1.2 EOR
%   O:3.0/12  FEEDER_EN  "feeder bowl enable" %
%   O:1.2  FEED_BOOL_SPD_OUT  "Feeder Bowl Speed Analog Output" %
% Rung: 8 %
SOR MOV N7:34 O:1.3 EOR
%   N7:34  HOPPER_SPD %
%   O:1.3  HOPPER_SPD_OUT  "Hopper Speed Analog Output" %
% Rung: 9 %
SOR XIO O:3.0/13 MOV 0 O:1.3 EOR
%   O:3.0/13  HOPPER_EN  "feeder hopper enable" %
%   O:1.3  HOPPER_SPD_OUT  "Hopper Speed Analog Output" %
% Rung: 10 %
SOR MUL N7:18 F8:0 O:1.0 EOR
%   N7:18  RECERK_SPD %
%   O:1.0  RECERK_CNV_SPD_OUT  "Recirculation Conveyor Speed Analog Output" %
% Rung: 11 %
SOR XIO O:0.0/8 MOV 0 O:1.0 EOR
%   O:0.0/8  BOT_CONV  "enable" %
%   O:1.0  RECERK_CNV_SPD_OUT  "Recirculation Conveyor Speed Analog Output" %
% Rung: 12 %
SOR XIC B3:2/4 MOV N7:52 O:1.0 EOR
%   B3:2/4  "override recerk conveyor speed" %
%   O:1.0  RECERK_CNV_SPD_OUT  "Recirculation Conveyor Speed Analog Output" %
% Rung: 13 %
SOR END EOR

LADDER 16 "TOTALCOUNT"
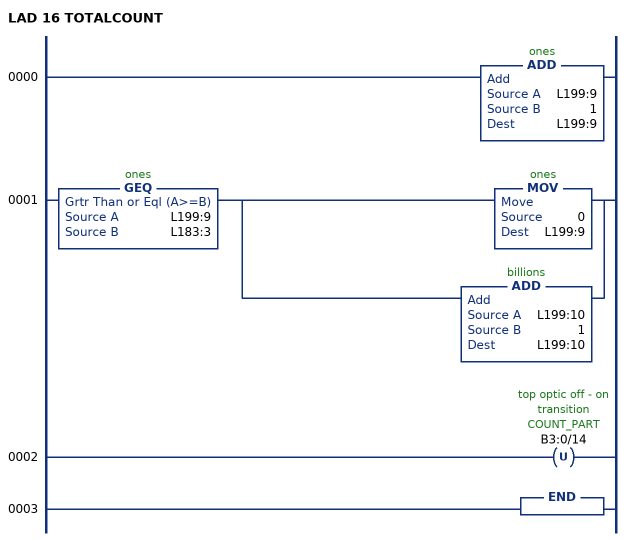
% Rung: 0 %
SOR ADD L199:9 1 L199:9 EOR
%   L199:9  "ones" %
% Rung: 1 %
SOR GEQ L199:9 L183:3 BST MOV 0 L199:9 NXB ADD L199:10 1 L199:10 BND EOR
%   L199:9  "ones" %
%   L183:3  "button state" %
%   L199:10  "billions" %
% Rung: 2 %
SOR OTU B3:0/14 EOR
%   B3:0/14  COUNT_PART  "top optic off - on transition" %
% Rung: 3 %
SOR END EOR

LADDER 18 "TESTTRIG1"
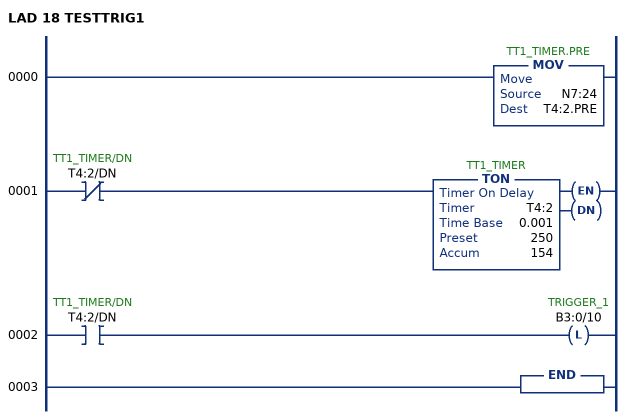
% Rung: 0 %
SOR MOV N7:24 T4:2.PRE EOR
%   T4:2  TT1_TIMER %
% Rung: 1 %
SOR XIO T4:2/DN TON T4:2 0.001 250 154 EOR
%   T4:2  TT1_TIMER %
% Rung: 2 %
SOR XIC T4:2/DN OTL B3:0/10 EOR
%   T4:2  TT1_TIMER %
%   B3:0/10  TRIGGER_1 %
% Rung: 3 %
SOR END EOR

LADDER 20 "TESTTRIG2"
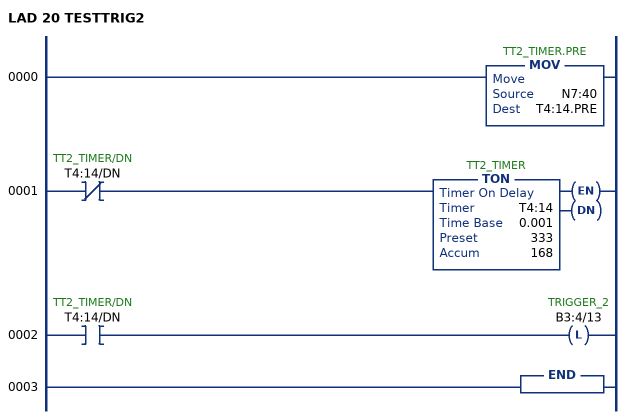
% Rung: 0 %
SOR MOV N7:40 T4:14.PRE EOR
%   T4:14  TT2_TIMER %
% Rung: 1 %
SOR XIO T4:14/DN TON T4:14 0.001 333 168 EOR
%   T4:14  TT2_TIMER %
% Rung: 2 %
SOR XIC T4:14/DN OTL B3:4/13 EOR
%   T4:14  TT2_TIMER %
%   B3:4/13  TRIGGER_2 %
% Rung: 3 %
SOR END EOR

LADDER 24 "SKIPPED"
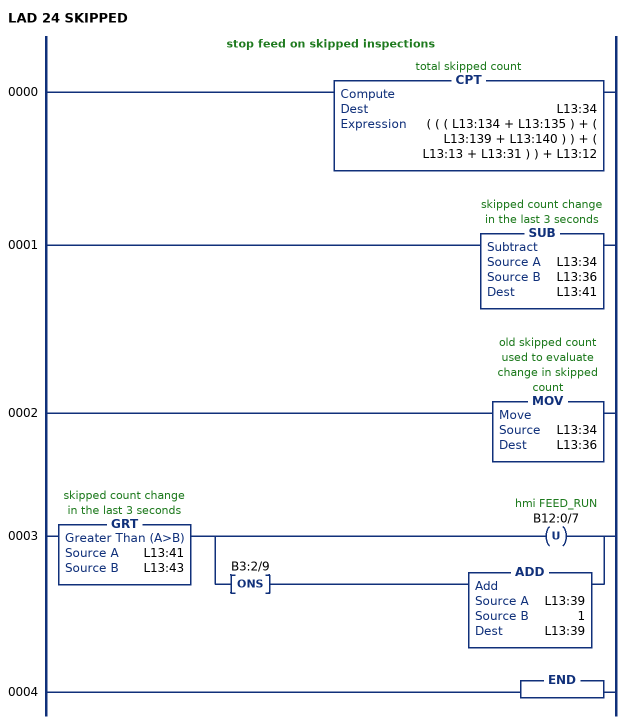
% Rung: 0 %
% TITLE: stop feed on skipped inspections %
SOR CPT L13:34 " ( ( ( L13:134 + L13:135 ) + ( L13:139 + L13:140 ) ) + ( L13:13 + L13:31 ) ) + L13:12 " EOR
%   L13:34  "total skipped count" %
%   L13:134  "too wide bottom" %
%   L13:135  "too close bottom" %
%   L13:139  "too close top count" %
%   L13:140  "too wide top count" %
%   L13:13  SKIP1  "skipped 1 count" %
%   L13:31  SKIP5  "skipped 5 count" %
%   L13:12  SKIP6  "skipped 6 count" %
% Rung: 1 %
SOR SUB L13:34 L13:36 L13:41 EOR
%   L13:34  "total skipped count" %
%   L13:36  "old skipped count used to evaluate change in skipped count" %
%   L13:41  "skipped count change in the last 3 seconds" %
% Rung: 2 %
SOR MOV L13:34 L13:36 EOR
%   L13:34  "total skipped count" %
%   L13:36  "old skipped count used to evaluate change in skipped count" %
% Rung: 3 %
SOR GRT L13:41 L13:43 BST OTU B12:0/7 NXB ONS B3:2/9 ADD L13:39 1 L13:39 BND EOR
%   L13:41  "skipped count change in the last 3 seconds" %
%   L13:43  "trigger count 1" %
%   B12:0/7  FEED_RUN  "hmi" %
% Rung: 4 %
SOR END EOR

LADDER 70 "ALIGNFAILS"    % normal %
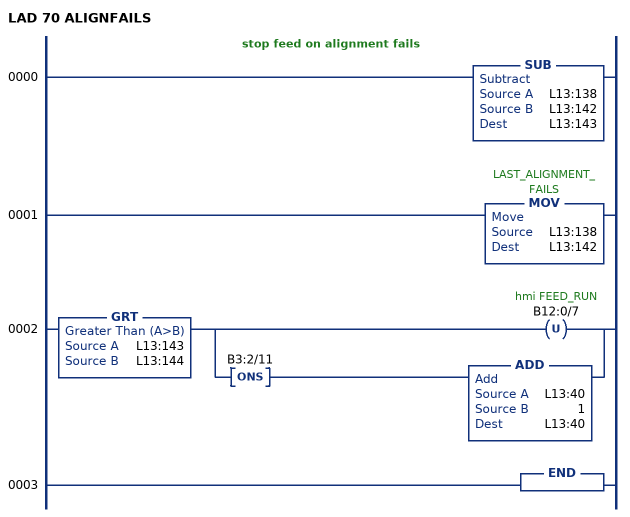
% Rung: 0 %
% TITLE: stop feed on alignment fails %
SOR SUB L13:138 L13:142 L13:143 EOR
%   L13:138  "alignment fail counts" %
%   L13:142  LAST_ALIGNMENT_FAILS %
% Rung: 1 %
SOR MOV L13:138 L13:142 EOR
%   L13:138  "alignment fail counts" %
%   L13:142  LAST_ALIGNMENT_FAILS %
% Rung: 2 %
SOR GRT L13:143 L13:144 BST OTU B12:0/7 NXB ONS B3:2/11 ADD L13:40 1 L13:40 BND EOR
%   B12:0/7  FEED_RUN  "hmi" %
% Rung: 3 %
SOR END EOR

LADDER 80 "HSC BOT"
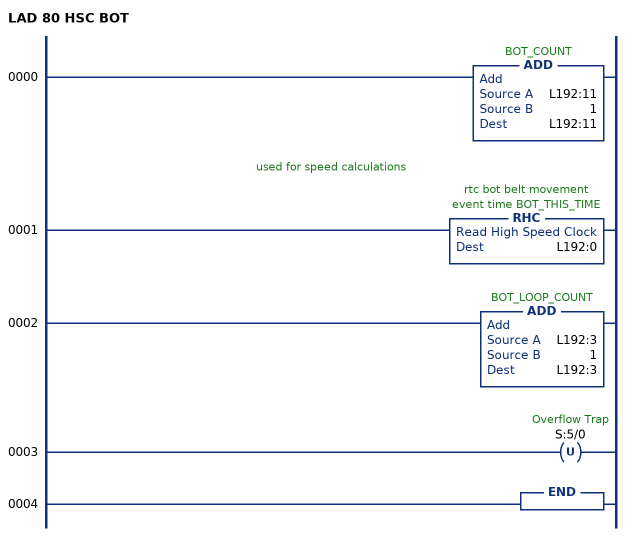
% Rung: 0 %
SOR ADD L192:11 1 L192:11 EOR
%   L192:11  BOT_COUNT %
% Rung: 1 %
% used for speed calculations %
SOR RHC L192:0 EOR
%   L192:0  BOT_THIS_TIME  "rtc bot belt movement event time" %
% Rung: 2 %
SOR ADD L192:3 1 L192:3 EOR
%   L192:3  BOT_LOOP_COUNT %
% Rung: 3 %
SOR OTU S:5/0 EOR
%   S:5/0  "Overflow Trap" %
% Rung: 4 %
SOR END EOR

LADDER 100 "1 MS STI"    % high speed %
